FUNCTION_BLOCK FB_VisuControl EXTENDS FB_UniversalVisu
VAR
END_VAR

bBackupRestoreDisabled := TRUE;
SUPER^();

METHOD PROTECTED  MS_Emergency
;
END_METHOD

END_FUNCTION_BLOCK

(* stored: Version 1.1.0.1, ProductVersion 3.1.4024.9
   POU FB_VisuControl: Id {8c70c37d-b6ba-41ef-bc85-65e1cd7c2b85}, SpecialFunc None
   Method MS_Emergency: Id {1f1e2364-c181-48ca-97b9-c39b4fa5dd63} *)
